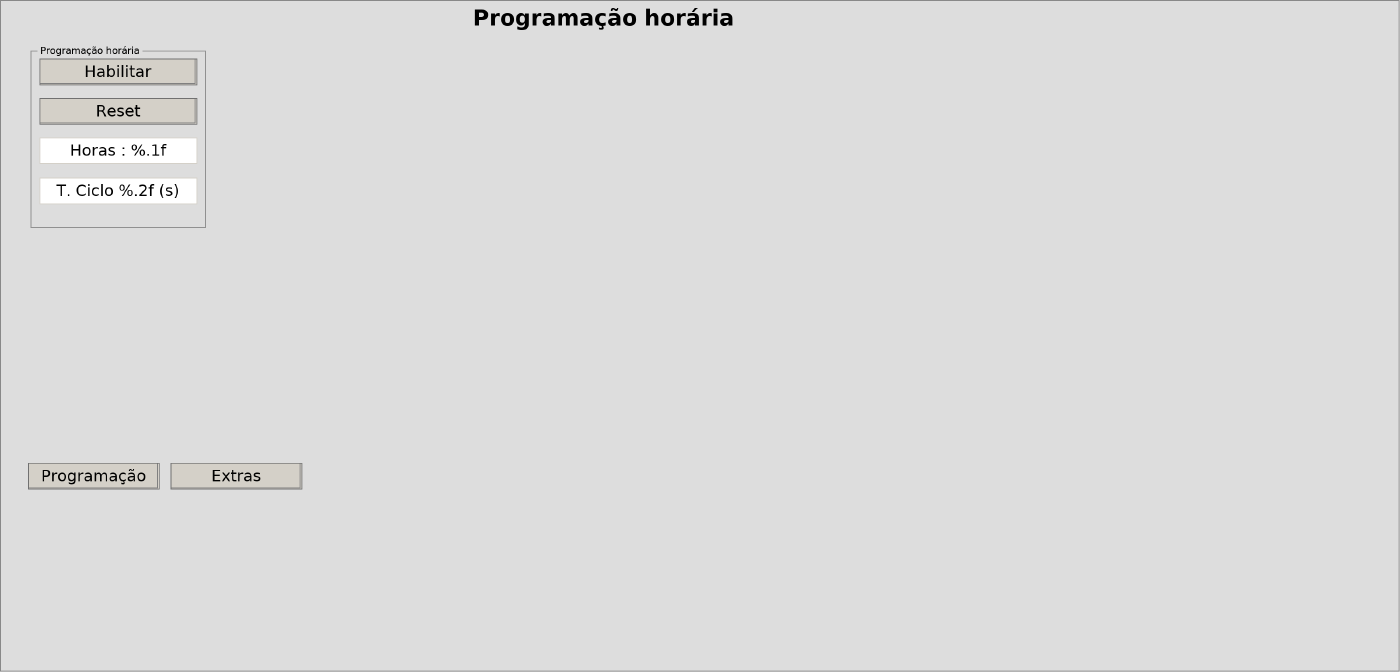
VISUALIZATION FuncoesExtras  // 1600x768
    Label (500,5 380x30), "Programação horária"
    Button (32,529 150x30), "Programação"
        OnMouseClick: change screen: Visualization
    Button (195,529 150x30), "Extras"
        OnMouseClick: change screen: FuncoesExtras
    GroupBox (35,50 200x210), "Programação horária"
        Button (10,17 180x30), "Habilitar"
            toggle GVL_TimeMeter.enableTimeCount
        Button (10,62 180x30), "Reset"
            tap GVL_TimeMeter.resetTimeCount
        Textfield (10,107 180x30), "Horas : %.1f", text variable: GVL_TimeMeter.hourCounting
        Textfield (10,153 180x30), "T. Ciclo %.2f (s)", text variable: GVL_TimeMeter.currTaskTime
END_VISUALIZATION

(* stored: Version 1.1.0.1, ProductVersion 3.1.4024.11
   Visu FuncoesExtras: Id {3b2c49e9-d451-436f-9bd8-7acdf8ee1440} *)
